// TIA Portal V20 export
DATA_BLOCK "SBK1"   // DB285
// stored: MemoryReserve 100
   VAR
      "X1-1 EMO01 CH.A" : Bool;
      "X2-1 EMO02 CH.A" : Bool;
      "X3-1 EMO03 CH.A" : Bool;
      "X4-1 EMO04 CH.A" : Bool;
      "X1-2 EMO01 CH.B" : Bool;
      "X2-2 EMO02 CH.B" : Bool;
      "X3-2 EMO03 CH.B" : Bool;
      "X4-2 EMO04 CH.B" : Bool;
   END_VAR
BEGIN
END_DATA_BLOCK
